// Mitsubishi GX Works2 project: solvvNpress_2   PLC: Q03UDV

PROGRAM MAIN
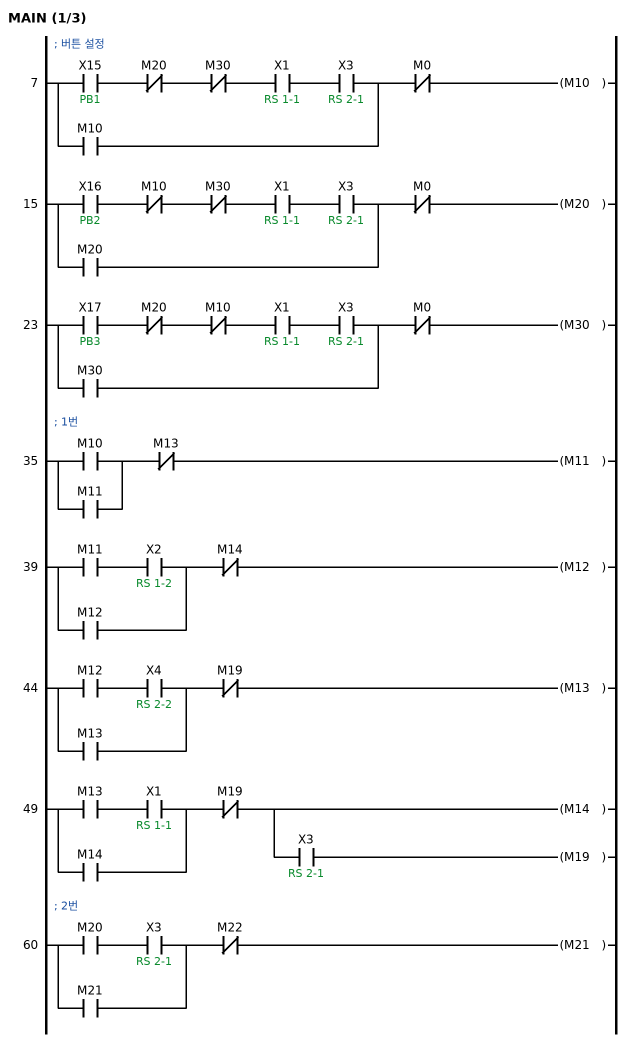
; 버튼 설정
7     LD      X15  ; PB1
      ANI     M20
      ANI     M30
      AND     X1  ; RS 1-1
      AND     X3  ; RS 2-1
      OR      M10
      ANI     M0
      OUT     M10
15    LD      X16  ; PB2
      ANI     M10
      ANI     M30
      AND     X1  ; RS 1-1
      AND     X3  ; RS 2-1
      OR      M20
      ANI     M0
      OUT     M20
23    LD      X17  ; PB3
      ANI     M20
      ANI     M10
      AND     X1  ; RS 1-1
      AND     X3  ; RS 2-1
      OR      M30
      ANI     M0
      OUT     M30
; 1번
35    LD      M10
      OR      M11
      ANI     M13
      OUT     M11
39    LD      M11
      AND     X2  ; RS 1-2
      OR      M12
      ANI     M14
      OUT     M12
44    LD      M12
      AND     X4  ; RS 2-2
      OR      M13
      ANI     M19
      OUT     M13
49    LD      M13
      AND     X1  ; RS 1-1
      OR      M14
      ANI     M19
      OUT     M14
      AND     X3  ; RS 2-1
      OUT     M19
; 2번
60    LD      M20
      AND     X3  ; RS 2-1
      OR      M21
      ANI     M22
      OUT     M21
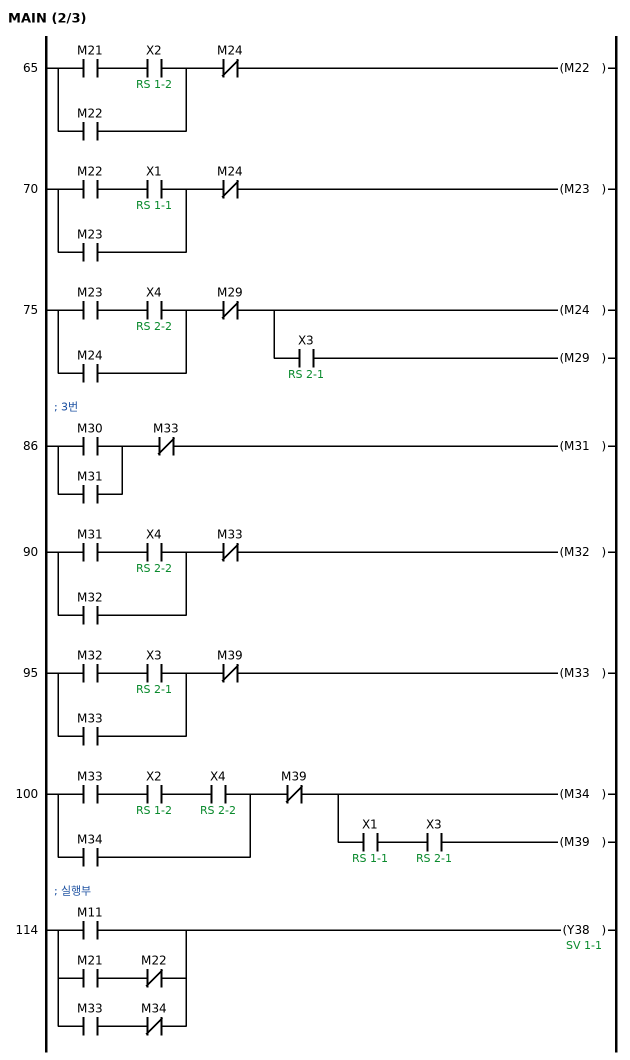
65    LD      M21
      AND     X2  ; RS 1-2
      OR      M22
      ANI     M24
      OUT     M22
70    LD      M22
      AND     X1  ; RS 1-1
      OR      M23
      ANI     M24
      OUT     M23
75    LD      M23
      AND     X4  ; RS 2-2
      OR      M24
      ANI     M29
      OUT     M24
      AND     X3  ; RS 2-1
      OUT     M29
; 3번
86    LD      M30
      OR      M31
      ANI     M33
      OUT     M31
90    LD      M31
      AND     X4  ; RS 2-2
      OR      M32
      ANI     M33
      OUT     M32
95    LD      M32
      AND     X3  ; RS 2-1
      OR      M33
      ANI     M39
      OUT     M33
100   LD      M33
      AND     X2  ; RS 1-2
      AND     X4  ; RS 2-2
      OR      M34
      ANI     M39
      OUT     M34
      AND     X1  ; RS 1-1
      AND     X3  ; RS 2-1
      OUT     M39
; 실행부
114   LD      M11
      LD      M21
      ANI     M22
      ORB
      LD      M33
      ANI     M34
      ORB
      OUT     Y38  ; SV 1-1
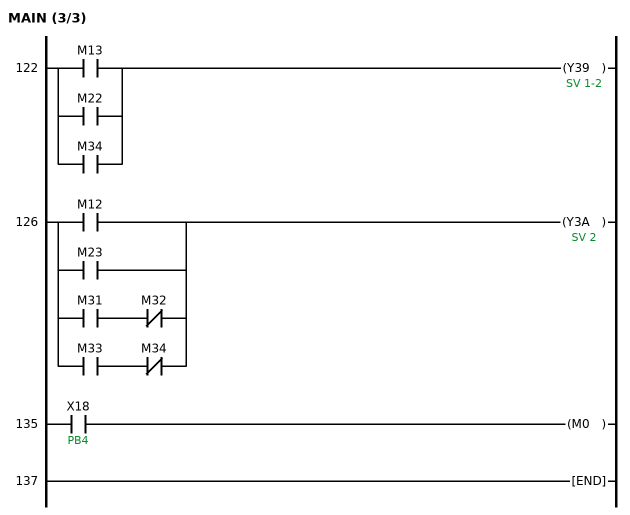
122   LD      M13
      OR      M22
      OR      M34
      OUT     Y39  ; SV 1-2
126   LD      M12
      OR      M23
      LD      M31
      ANI     M32
      ORB
      LD      M33
      ANI     M34
      ORB
      OUT     Y3A  ; SV 2
135   LD      X18  ; PB4
      OUT     M0
137   END
END_PROGRAM

// device comments not shown above
X19  ; PB5
Y30  ; LAMP1
Y31  ; LAMP2
Y3B  ; SV 3
